# EPICS autosave request: iocBoot/ioc13idd_DAC_XPS/auto_settings.req
file "userArrayCalcs10_settings.req",   P=$(P)
file "userCalcOuts10_settings.req",     P=$(P)
file "userStringCalcs10_settings.req",  P=$(P)
file "userStringSeqs10_settings.req",   P=$(P)
file "userTransforms10_settings.req",   P=$(P)
file "CARS_motor_settings.req",         P=$(P), M=m81
file "CARS_motor_settings.req",         P=$(P), M=m82
file "CARS_motor_settings.req",         P=$(P), M=m83
file "CARS_motor_settings.req",         P=$(P), M=m84
